RoboDK station: objects_in_scene.rdk

Station scene. Poses are relative to the parent item; angles as X-Y-Z fixed-axis rotations.
  - frame Origin at (0, 0, 0) mm
  - frame Cameras at (0, 1000, 0) mm
    - frame Camera_1 at (-2118.36, -747.6, 4441.52) mm, rotated rx -180 ry -60 rz 0 deg
    - frame Camera_2 at (3225.8, -873, 4530.73) mm, rotated rx -180 ry 60 rz 0 deg
  - frame Walls at (0, 2000, 0) mm
    - frame Left_Wall_1 at (-2120.9, -1847.6, 4581.52) mm, rotated rx 0 ry 90 rz 0 deg
    - frame Left_Wall_2 at (-2476.5, -1933.33, 2295.53) mm, rotated rx 0 ry 90 rz 0 deg
    - frame Right_Wall_1 at (3289.3, -1949.2, 1460.5) mm, rotated rx 0 ry -90 rz 0 deg
    - frame Right_Wall_2 at (3289.3, -1974.6, 4022.72) mm, rotated rx 0 ry -90 rz 0 deg
  - frame Chairs at (0, 3000, 0) mm
    - frame Chair_1 at (-127, -2918, 3492) mm, rotated rx 0 ry -90 rz -19.2 deg
    - frame Chair_2 at (-127, -2917.45, 4114.8) mm, rotated rx 0 ry -90 rz -19.2 deg
    - frame Chair_3 at (1009.65, -2917.45, 4314.8) mm, rotated rx 0 ry 90 rz 19.2 deg
    - frame Chair_4 at (1009.65, -2917.45, 3692.5) mm, rotated rx 0 ry 90 rz 19.2 deg
  - frame Waypoints at (0, 4000, 0) mm
    - frame Waypoint_1 at (515, -3850, 1644) mm, rotated rx 0 ry -90 rz -90 deg
    - frame Waypoint_2 at (2294, -3850, 3950) mm, rotated rx 90 ry 0 rz -180 deg
    - frame Waypoint_3 at (515, -3850, 6032) mm, rotated rx 0 ry 90 rz 90 deg
    - frame Waypoint_4 at (-1714, -3850, 3950) mm, rotated rx -90 ry 0 rz 0 deg
